// TIA Portal V21 export
VAR_GLOBAL   // PLC tag table "K_MacchinaARicetta"
END_VAR
VAR_GLOBAL CONSTANT   // user constants
   K_MacchinaARicetta_SterilizzatoreTubo : Int := 1;   // Sterilisatorschlauch / Sterilizertube / Esterilizador tubo / Stérilisateurtube / Sterilizzatoretubo
END_VAR
